RoboDK station: Assistive_UR5e_nou (còpia).rdk

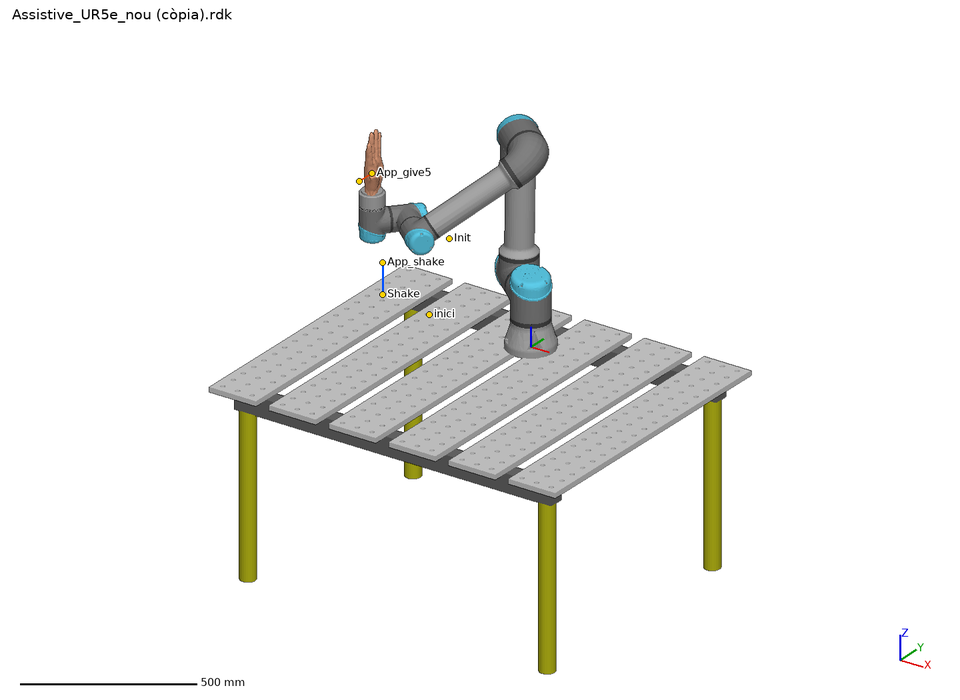
[picture v0: the station drawn from its stored meshes, robots at their saved joint values, targets as dots, program paths as lines]
Station Assistive_UR5e_nou (saved by RoboDK 5.9.2). Poses are relative to the parent item; angles as X-Y-Z fixed-axis rotations.
  - frame UR5e Base at (0, 0, 0) mm
    - robot UR5e: 6 axes, payload 5 kg, reach 850 mm, repeatability 0.03 mm, weight 18.4 kg
        modified DH rows (alpha deg, a mm, theta deg, d mm): 0, 0, 0, 162.5; 90, 0, 180, 0; 0, 425, 0, 0; 0, 392.25, 0, 133.3; -90, 0, 0, 99.7; 90, 0, 180, 99.6
        joint limits [-360, -360, -360, -360, -360, -360] to [360, 360, 360, 360, 360, 360]; home [0, -90, -90, 0, 90, 0]; saved at [-130.679, -89.195, -122.013, 301.208, -90, -119.321]
      - tool Hand, TCP at (0, 0, 50) mm, size 54.8 x 155.9 x 193.5 mm, geometry from Hand.stl
  - frame World at (0, 0, 0) mm
    - object Table at (0, 0, 0) mm, size 1193.8 x 965.2 x 609.6 mm, geometry from welding_table.sld
    - target Init (Cartesian target) at (0, -400, 500) mm, rotated rx 90 ry 0 rz 0 deg; joints [-57.836, -65.392, -107.167, 172.559, -57.836, 0] of UR5e
    - target App_shake (joint target) at (-300, -300, 300) mm, rotated rx 90 ry 0 rz 0 deg; joints [-129.97, -84.968, -123.366, -151.667, -129.97, 0] of UR5e
    - target Shake (joint target) at (-300, -300, 200) mm, rotated rx 90 ry 0 rz 0 deg; joints [-129.97, -95.332, -131.473, -133.195, -129.97, 0] of UR5e
    - target App_give5 (joint target) at (-380.86, -238.62, 533.82) mm, rotated rx 0 ry 0 rz 90 deg; joints [-130.679, -89.195, -122.013, 301.208, -90, 130.679] of UR5e
    - target Give5 (joint target) at (-380.86, -300, 533.82) mm, rotated rx 0 ry 0 rz 90 deg; joints [-125.814, -94.091, -116.939, 301.03, -90, 125.814] of UR5e
    - target inici (Cartesian target) at (0, -500, 300) mm, rotated rx 90 ry 0 rz 0 deg; joints [-292.36, 20.37, -121.299, 100.929, -292.36, 0] of UR5e
    - target ventilar (Cartesian target) at (-380.86, -238.62, 533.82) mm, rotated rx 0 ry 0 rz -160 deg; joints [14.815, 20.403, -90.958, 160.555, -90, 95.185] of UR5e
    - target abaix (Cartesian target) at (-380.86, -238.62, 533.82) mm, rotated rx -4.31 ry -30.91 rz -164.48 deg; joints [-136.691, -101.772, -111.73, 329.548, -107.784, 245.158] of UR5e
  - program Init (3 instructions, listed below)
  - program Hand_shake (5 instructions, listed below)
  - program Give_me_5! (5 instructions, listed below)
  - program MainProgram (4 instructions, listed below)
  - Python program Assistive_hand_SW_nova_funcio (listed below)
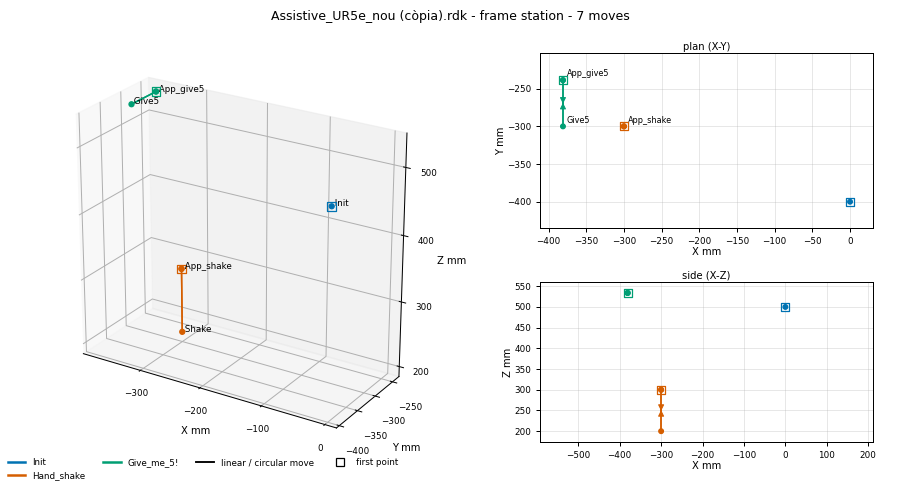
[picture p0: tool path of Assistive_UR5e_nou (còpia).rdk in frame station, 7 of 7 moves have a stored position in this frame; points joined in program order, loops and branches not executed]

--- program Init (robot UR5e) ---
  Est. Ref.: UR5e Base
  Est. herr: Hand
  MoveJ (Init)

--- program Hand_shake (robot UR5e) ---
  Est. Ref.: UR5e Base
  Est. herr: Hand
  MoveL (App_shake)
  MoveL (Shake)
  MoveL (App_shake)

--- program Give_me_5! (robot UR5e) ---
  Est. Ref.: UR5e Base
  Est. herr: Hand
  MoveL (App_give5)
  MoveL (Give5)
  MoveL (App_give5)

--- program MainProgram (robot UR5e) ---
  Llamar Init
  Llamar Hand_shake
  Llamar Give_me_5!
  Llamar Init

--- Python program Assistive_hand_SW_nova_funcio ---
from robodk.robolink import *
from robodk.robomath import *

# Robot setup
RDK = Robolink()
robot = RDK.Item("UR5e")
base = RDK.Item("UR5e Base")
tool = RDK.Item('Hand')
Init_target = RDK.Item('Init')
App_shake_target = RDK.Item('App_shake')
Shake_target = RDK.Item('Shake')
App_give5_target = RDK.Item('App_give5')
Give5_target = RDK.Item('Give5')
#Punts que hem definit nosaltres (nous)
inici_target = RDK.Item('inici')
ventilar_target = RDK.Item('ventilar')
abaix_target = RDK.Item('abaix')

robot.setPoseFrame(base)
robot.setPoseTool(tool)
robot.setSpeed(20)

def Init():
    print("Init")
    robot.MoveL(Init_target, True)
    print("Init_target REACHED")

def Hand_shake():
    print("Hand Shake")
    robot.MoveL(App_shake_target, True)
    robot.MoveL(Shake_target, True)
    robot.MoveL(App_shake_target, True)
    print("Hand Shake FINISHED")

def Give_me_5():
    print("Give me 5!")
    robot.MoveL(App_give5_target, True)
    robot.MoveL(Give5_target, True)
    robot.MoveL(App_give5_target, True)
    print("Give me 5! FINISHED")

def nova_funcio():
    print("Quina calor!")
    robot.MoveL(inici_target, True)
    robot.MoveL(ventilar_target, True)
    robot.MoveL(abaix_target, True)
    robot.MoveL(ventilar_target, True)
    robot.MoveL(abaix_target, True)
    robot.MoveL(ventilar_target, True)
    print("nova_funcio FINISHED")

# Main function
#def main():
  #  Init()
  #  Hand_shake()
   # Give_me_5()
   # Init()

# Main function
def main():
    nova_funcio()


if __name__ == "__main__":
    main()
